RESOURCE_TYPE FlexPRET
  (* Standard: 61499-2 *)
  (* Version 0.1, 2016-00-28, hpea485, UOA *)
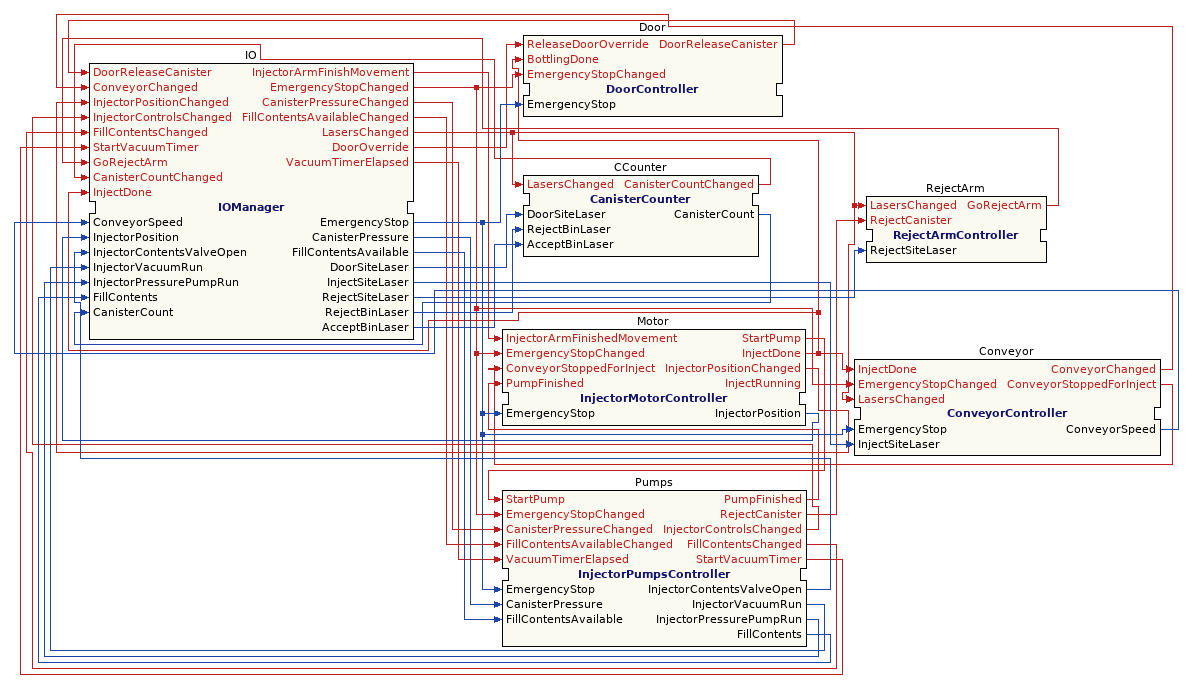
  FBS
    IO : IOManager;
    CCounter : CanisterCounter;
    Door : DoorController;
    Conveyor : ConveyorController;
    RejectArm : RejectArmController;
    Pumps : InjectorPumpsController;
    Motor : InjectorMotorController;
  END_FBS
  EVENT_CONNECTIONS
    IO.InjectorArmFinishMovement TO Motor.InjectorArmFinishedMovement;
    IO.EmergencyStopChanged TO Door.EmergencyStopChanged;
    IO.EmergencyStopChanged TO Conveyor.EmergencyStopChanged;
    IO.EmergencyStopChanged TO Motor.EmergencyStopChanged;
    IO.EmergencyStopChanged TO Pumps.EmergencyStopChanged;
    IO.CanisterPressureChanged TO Pumps.CanisterPressureChanged;
    IO.FillContentsAvailableChanged TO Pumps.FillContentsAvailableChanged;
    IO.LasersChanged TO CCounter.LasersChanged;
    IO.LasersChanged TO RejectArm.LasersChanged;
    IO.LasersChanged TO Conveyor.LasersChanged;
    IO.DoorOverride TO Door.ReleaseDoorOverride;
    IO.VacuumTimerElapsed TO Pumps.VacuumTimerElapsed;
    CCounter.CanisterCountChanged TO IO.CanisterCountChanged;
    Door.DoorReleaseCanister TO IO.DoorReleaseCanister;
    Conveyor.ConveyorChanged TO IO.ConveyorChanged;
    Conveyor.ConveyorStoppedForInject TO Motor.ConveyorStoppedForInject;
    RejectArm.GoRejectArm TO IO.GoRejectArm;
    Pumps.PumpFinished TO Motor.PumpFinished;
    Pumps.RejectCanister TO RejectArm.RejectCanister;
    Pumps.InjectorControlsChanged TO IO.InjectorControlsChanged;
    Pumps.FillContentsChanged TO IO.FillContentsChanged;
    Pumps.StartVacuumTimer TO IO.StartVacuumTimer;
    Motor.StartPump TO Pumps.StartPump;
    Motor.InjectDone TO Door.BottlingDone;
    Motor.InjectDone TO Conveyor.InjectDone;
    Motor.InjectDone TO IO.InjectDone;
    Motor.InjectorPositionChanged TO IO.InjectorPositionChanged;
  END_CONNECTIONS
  DATA_CONNECTIONS
    IO.EmergencyStop TO Door.EmergencyStop;
    IO.EmergencyStop TO Conveyor.EmergencyStop;
    IO.EmergencyStop TO Motor.EmergencyStop;
    IO.EmergencyStop TO Pumps.EmergencyStop;
    IO.CanisterPressure TO Pumps.CanisterPressure;
    IO.FillContentsAvailable TO Pumps.FillContentsAvailable;
    IO.DoorSiteLaser TO CCounter.DoorSiteLaser;
    IO.InjectSiteLaser TO Conveyor.InjectSiteLaser;
    IO.RejectSiteLaser TO RejectArm.RejectSiteLaser;
    IO.RejectBinLaser TO CCounter.RejectBinLaser;
    IO.AcceptBinLaser TO CCounter.AcceptBinLaser;
    CCounter.CanisterCount TO IO.CanisterCount;
    Conveyor.ConveyorSpeed TO IO.ConveyorSpeed;
    Pumps.InjectorContentsValveOpen TO IO.InjectorContentsValveOpen;
    Pumps.InjectorVacuumRun TO IO.InjectorVacuumRun;
    Pumps.InjectorPressurePumpRun TO IO.InjectorPressurePumpRun;
    Pumps.FillContents TO IO.FillContents;
    Motor.InjectorPosition TO IO.InjectorPosition;
  END_CONNECTIONS
END_RESOURCE_TYPE
